Yaskawa INFORM job: ADD-TACK-BY-TEACH-IN-2-S2.JBI

/JOB
//NAME ADD-TACK-BY-TEACH-IN-2-S2
//POS
///NPOS 0,0,0,0,0,0
//INST
///DATE 2018/11/22 18:37
///ATTR SC,RW
///GROUP1 RB1,BS1
///GROUP2 ST2
NOP
END
